// TIA Portal project "converge_station_project" (V15.1)
// Vorlageprojekt für das Buch mit Zielsystem S7-1200

(* hardware
DEVICE "S7-1200-Station_1"  S7-1200 Station
   slot 0: "Baugruppenträger_0"  Rack  V1.0
   slot 1: "PLC_1"  CPU 1211C DC/DC/DC  6ES7 211-1AE40-0XB0  V4.1
*)

// ===== PLC "PLC_1"  CPU 1211C DC/DC/DC =====

VAR_GLOBAL   // PLC tag table "Standard-Variablentabelle"
   "Conveyor 1" AT %A0.0 : Bool;
   "START" AT %I0.5 : Bool;
   "Unload 1" AT %Q0.2 : Bool;
   "Load 1" AT %Q0.1 : Bool;
   "Exit conveyor" AT %Q1.2 : Bool;
   "Conveyor 2" AT %Q0.5 : Bool;
   "At entry 2" AT %I0.1 : Bool;
   "Load 2" AT %Q0.6 : Bool;
   "At entry 1" AT %I0.0 : Bool;
   "At exit" AT %I0.4 : Bool;
   "At transfer 1" AT %I0.2 : Bool;
   "At transfer 2" AT %I0.3 : Bool;
   "Transfer right 1" AT %Q0.3 : Bool;
   "Transfer left 1" AT %Q0.4 : Bool;
   "Transfer right 2" AT %Q1.0 : Bool;
   "Transfer left 2" AT %Q1.1 : Bool;
   "Counter" AT %QD30 : DInt;
   "At exit M" AT %M0.0 : Bool;
END_VAR

// folder: System blocks/Program resources

DATA_BLOCK "IEC_Timer_0_DB"   // DB1
{ S7_Optimized_Access := 'TRUE' }
AUTHOR : Simatic
FAMILY : IEC
NAME : IEC_TMR
VERSION : 1.0
// stored: InstanceOfName IEC_TIMER
"IEC_TIMER"
BEGIN
END_DATA_BLOCK

// folder: (top level)

FUNCTION "MHJ-PLC-Lab-Function-S71200" : Void   // FC9000, SCL
{ S7_Optimized_Access := 'TRUE' }
VERSION : 0.1
   VAR_TEMP
      rdTimeReturn : Int;
      outputTime : DTL;
      SyncVal : Byte;
      forVal : Int;
      forVal_2 : Int;
      Value : Byte;
   END_VAR
   VAR CONSTANT
      CompVal : Byte := 16#34;
      Value_01 : Byte := 16#11;
      Value_01_DW : DWord := 16#A165_D992;
      Value_02_DW : DWord := 16#58BE_4401;
   END_VAR
BEGIN

   #Value:=PEEK(area := 16#82,
        dbNumber := 0,
        byteOffset := 511);
   #Value := #Value + 1;

   POKE(area := 16#82,
        dbNumber := 0,
        byteOffset := 511,
        value := #Value);

   POKE(area:=16#81,
        dbNumber:=0,
        byteOffset:=1016,
        value:=#Value_01_DW);
   POKE(area := 16#81,
        dbNumber := 0,
        byteOffset := 1020,
        value := #Value_02_DW);

   POKE(area := 16#81,
        dbNumber := 0,
        byteOffset := 511,
        value := B#16#00);

   FOR #forVal := 0 TO 120 DO
       FOR #forVal_2:=0 TO 10 DO
           #rdTimeReturn:=RD_SYS_T(#outputTime);
           #rdTimeReturn := WR_SYS_T(#outputTime);
           #rdTimeReturn := RD_SYS_T(#outputTime);
           #rdTimeReturn := WR_SYS_T(#outputTime);
       END_FOR;
       #SyncVal:= PEEK(area := 16#81,
                      dbNumber := 0,
                      byteOffset := 511);
       IF #SyncVal = #CompVal THEN
          GOTO M_1;
       END_IF;
   END_FOR;
   RETURN;

   M_1:
   POKE(area := 16#81,
        dbNumber := 0,
        byteOffset := 511,
        value := B#16#0);
END_FUNCTION

ORGANIZATION_BLOCK "Main"   // OB1, LAD, ProgramCycle
TITLE = "Main Program Sweep (Cycle)"
{ S7_Optimized_Access := 'TRUE' }
VERSION : 0.1
   VAR_INPUT
      Initial_Call : Bool;   // Initial call of this OB
      Remanence : Bool;   // =True, if remanent data are available
   END_VAR
   VAR_TEMP   // added for the SCL form of the ladder/FBD networks
      _w1 : Bool;
   END_VAR
BEGIN

REGION Network 1: Konnektierungsbaustein für PLC-Lab
   // Im Netzwerk 1 wird der Konnektierungsbaustein für PLC-Lab aufgerufen.
   // Dieser Aufruf darf nicht entfernt werden!
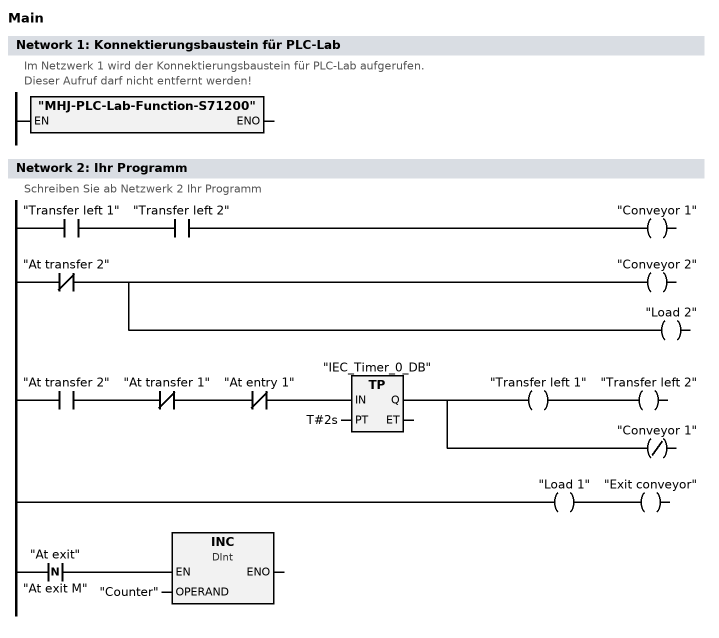
   RUNG wire#powerrail
      "MHJ-PLC-Lab-Function-S71200"()
   END_RUNG
   // the same network as SCL:
   "MHJ-PLC-Lab-Function-S71200"();
END_REGION

REGION Network 2: Ihr Programm
   // Schreiben Sie ab Netzwerk 2 Ihr Programm
   "Conveyor 1" := "Transfer left 1" AND "Transfer left 2";
   "Conveyor 2" := NOT "At transfer 2";
   "Load 2" := NOT "At transfer 2";
   "IEC_Timer_0_DB".TP(IN := "At transfer 2" AND NOT "At transfer 1" AND NOT "At entry 1", PT := T#2s);
   "Transfer left 1" := "IEC_Timer_0_DB".Q;
   "Transfer left 2" := "IEC_Timer_0_DB".Q;
   "Conveyor 1" := NOT "IEC_Timer_0_DB".Q;
   "Load 1" := TRUE;
   "Exit conveyor" := TRUE;
   #_w1 := NOT "At exit" AND "At exit M";   // falling edge of "At exit"
   "At exit M" := "At exit";
   IF #_w1 THEN "Counter" := "Counter" + 1; END_IF;
END_REGION
END_ORGANIZATION_BLOCK